FUNCTION_BLOCK FB_Controller_SFC
VAR_INPUT
	tm: REFERENCE TO FB_Timelimits; //S_Timeouts;
	//tm: FB_Timelimits; //S_Timeouts;
	IC: BOOL;
	Execute: BOOL;
	Ack: BOOL;
END_VAR
VAR_OUTPUT
	Ready: BOOL;
	Failure: BOOL;
	Done: BOOL;
END_VAR

END_FUNCTION_BLOCK

(* stored: Version 1.1.0.1, ProductVersion 3.1.4024.11
   POU FB_Controller_SFC: Id {b1eab9be-49a6-4397-bfc3-8676828bc4c5}, SpecialFunc None *)
